{attribute 'qualified_only' := ''}
{attribute 'strict' := ''}
{attribute 'to_string' := ''}
TYPE c3LnSwFaultCodes :
(
	InvalidTrafficControl := 0,
	InvalidOutputLane := 1
);
END_TYPE

(* stored: Version 1.1.0.1, ProductVersion 3.1.4024.6
   DUT c3LnSwFaultCodes: Id {60b2ad12-12a2-42b2-9379-7da31907beb0} *)
